//create working DB
DATA_BLOCK DB2101
STRUCT
START_SEQ:BYTE:=16#1;
END_SEQ:BYTE:=16#2;
SND_COMM_DB:WORD:=16#836;
WRT_COMM_DB:WORD:=16#837;
WRT_COMP_DB:WORD:=16#838;
DAT_RECV_DB:WORD:=16#839;
ACT_1:BOOL:=TRUE;
Mode_1:BOOL:=FALSE;
SND_DB_1:INT:=2102;
SND_ADD_1:INT:=0;
SND_LEN_1:INT:=6;
RCV_DB_1:INT:=2105;
RCV_ADD_1:INT:=0;
RCV_LEN_1:INT:=10;
WD_TIME_1:INT:=3000;
ACT_2:BOOL:=TRUE;
Mode_2:BOOL:=FALSE;
SND_DB_2:INT:=2104;
SND_ADD_2:INT:=0;
SND_LEN_2:INT:=10;
RCV_DB_2:INT:=2105;
RCV_ADD_2:INT:=10;
RCV_LEN_2:INT:=2;
WD_TIME_2:INT:=3000;
VBVer:WORD:=16#2B;   //配置文件版本号
END_STRUCT
BEGIN
END_DATA_BLOCK




//create SND_COMMAND DB
DATA_BLOCK DB2102
STRUCT
SlaveID_1:BYTE:=16#B;
FC_1:BYTE:=16#3;
START_ADD_1:WORD:=16#0;
DATA_NUM_1:WORD:=16#4;
CRC_1:WORD:=16#0;
END_STRUCT
BEGIN
END_DATA_BLOCK




//create WRT_COMMAND DB
DATA_BLOCK DB2103
STRUCT
SlaveID_2:BYTE:=16#B;
FC_2:BYTE:=16#10;
START_ADD_2:WORD:=16#4;
DATA_NUM_2:WORD:=16#1;
DATA_BYTE_2:WORD:=16#2;
DATA_2_1:WORD:=16#0;    //地址40005
CRC_2:WORD:=16#0;
END_STRUCT
BEGIN
END_DATA_BLOCK




//create WRT_COMPARE_COMMAND DB
DATA_BLOCK DB2104
STRUCT
SlaveID_2:BYTE:=16#B;
FC_2:BYTE:=16#10;
START_ADD_2:WORD:=16#4;
DATA_NUM_2:WORD:=16#1;
DATA_BYTE_2:WORD:=16#2;
DATA_NUM_2_1:WORD:=16#0;
CRC_2:WORD:=16#0;
END_STRUCT
BEGIN
END_DATA_BLOCK




//create DAT_COMMAND DB
DATA_BLOCK DB2105
STRUCT
Command_1_STATUS:WORD:=16#0;     //第1条命令的状态，0=正常，1=无响应，2=站号错误，3=命令错误，4=CRC校验错误
Command_1_DATA_1:WORD:=16#0;    //地址40001
Command_1_DATA_2:WORD:=16#0;    //地址40002
Command_1_DATA_3:WORD:=16#0;    //地址40003
Command_1_DATA_4:WORD:=16#0;    //地址40004
Command_2_STATUS:WORD:=16#0;     //第2条命令的状态，0=正常，1=无响应，2=站号错误，3=命令错误，4=CRC校验错误
END_STRUCT
BEGIN
END_DATA_BLOCK
